% RSLogix 500 project I2P JOB 12 B ALEXANDER_LOYND_BAK034.RSS, saved by version 10.00.00.00 %
PROJECT "ML06A"    % processor: Bul.1763 MicroLogix 1100 Series B %

PROGRAM FILES
  LAD 2   13 rungs

DATA FILES
  O0 OUTPUT  4 elements
  I1 INPUT  6 elements
  S2 STATUS  66 elements
  B3 BINARY  1 elements
  T4 TIMER  1 elements
  C5 COUNTER  1 elements
  R6 CONTROL  1 elements
  N7 INTEGER  1 elements
  F8 FLOAT  1 elements

LADDER 2
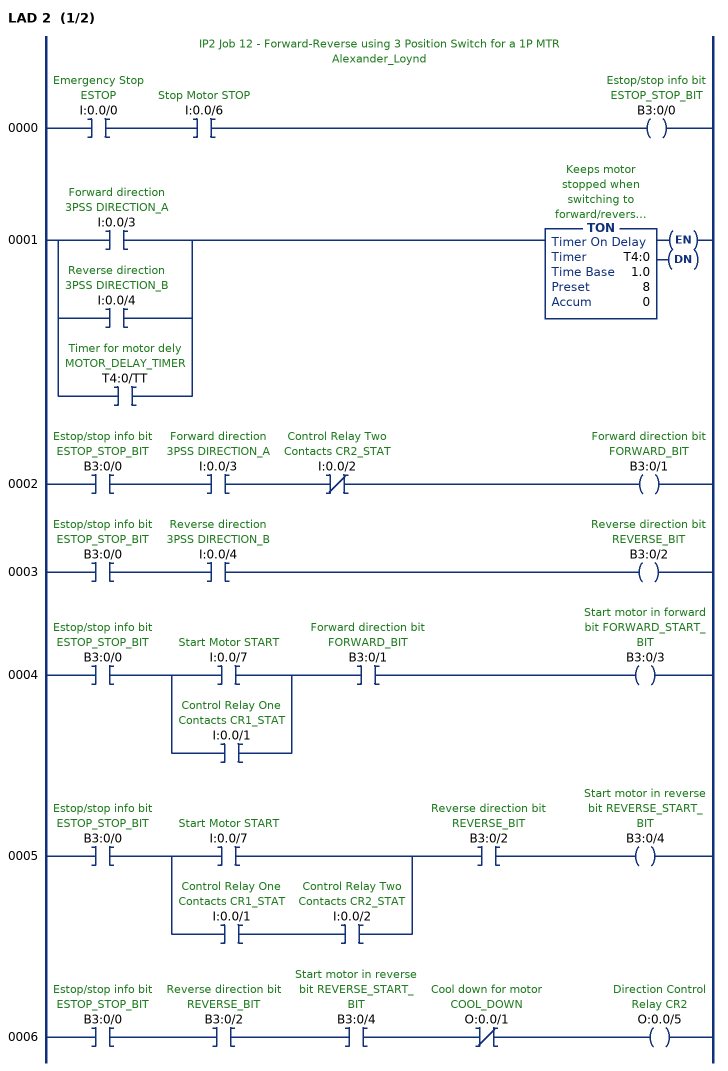
% Rung: 0 %
% IP2 Job 12 - Forward-Reverse using 3 Position Switch for a 1P MTR
% Alexander_Loynd %
SOR XIC I:0.0/0 XIC I:0.0/6 OTE B3:0/0 EOR
%   I:0.0/0  ESTOP  "Emergency Stop" %
%   I:0.0/6  STOP  "Stop Motor" %
%   B3:0/0  ESTOP_STOP_BIT  "Estop/stop info bit" %
% Rung: 1 %
SOR BST XIC I:0.0/3 NXB BST XIC I:0.0/4 NXB XIC T4:0/TT BND BND TON T4:0 1.0 8 0 EOR
%   I:0.0/3  DIRECTION_A  "Forward direction 3PSS" %
%   I:0.0/4  DIRECTION_B  "Reverse direction 3PSS" %
%   T4:0/TT  MOTOR_DELAY_TIMER  "Timer for motor dely" %
%   T4:0  TIME_ON_DELAY  "Keeps motor stopped when switching to forward/reverse" %
% Rung: 2 %
SOR XIC B3:0/0 XIC I:0.0/3 XIO I:0.0/2 OTE B3:0/1 EOR
%   B3:0/0  ESTOP_STOP_BIT  "Estop/stop info bit" %
%   I:0.0/3  DIRECTION_A  "Forward direction 3PSS" %
%   I:0.0/2  CR2_STAT  "Control Relay Two Contacts" %
%   B3:0/1  FORWARD_BIT  "Forward direction bit" %
% Rung: 3 %
SOR XIC B3:0/0 XIC I:0.0/4 OTE B3:0/2 EOR
%   B3:0/0  ESTOP_STOP_BIT  "Estop/stop info bit" %
%   I:0.0/4  DIRECTION_B  "Reverse direction 3PSS" %
%   B3:0/2  REVERSE_BIT  "Reverse direction bit" %
% Rung: 4 %
SOR XIC B3:0/0 BST XIC I:0.0/7 NXB XIC I:0.0/1 BND XIC B3:0/1 OTE B3:0/3 EOR
%   B3:0/0  ESTOP_STOP_BIT  "Estop/stop info bit" %
%   I:0.0/7  START  "Start Motor" %
%   I:0.0/1  CR1_STAT  "Control Relay One Contacts" %
%   B3:0/1  FORWARD_BIT  "Forward direction bit" %
%   B3:0/3  FORWARD_START_BIT  "Start motor in forward bit" %
% Rung: 5 %
SOR XIC B3:0/0 BST XIC I:0.0/7 NXB XIC I:0.0/1 XIC I:0.0/2 BND XIC B3:0/2 OTE B3:0/4 EOR
%   B3:0/0  ESTOP_STOP_BIT  "Estop/stop info bit" %
%   I:0.0/7  START  "Start Motor" %
%   I:0.0/1  CR1_STAT  "Control Relay One Contacts" %
%   I:0.0/2  CR2_STAT  "Control Relay Two Contacts" %
%   B3:0/2  REVERSE_BIT  "Reverse direction bit" %
%   B3:0/4  REVERSE_START_BIT  "Start motor in reverse bit" %
% Rung: 6 %
SOR XIC B3:0/0 XIC B3:0/2 XIC B3:0/4 XIO O:0.0/1 OTE O:0.0/5 EOR
%   B3:0/0  ESTOP_STOP_BIT  "Estop/stop info bit" %
%   B3:0/2  REVERSE_BIT  "Reverse direction bit" %
%   B3:0/4  REVERSE_START_BIT  "Start motor in reverse bit" %
%   O:0.0/1  COOL_DOWN  "Cool down for motor" %
%   O:0.0/5  CR2  "Direction Control Relay" %

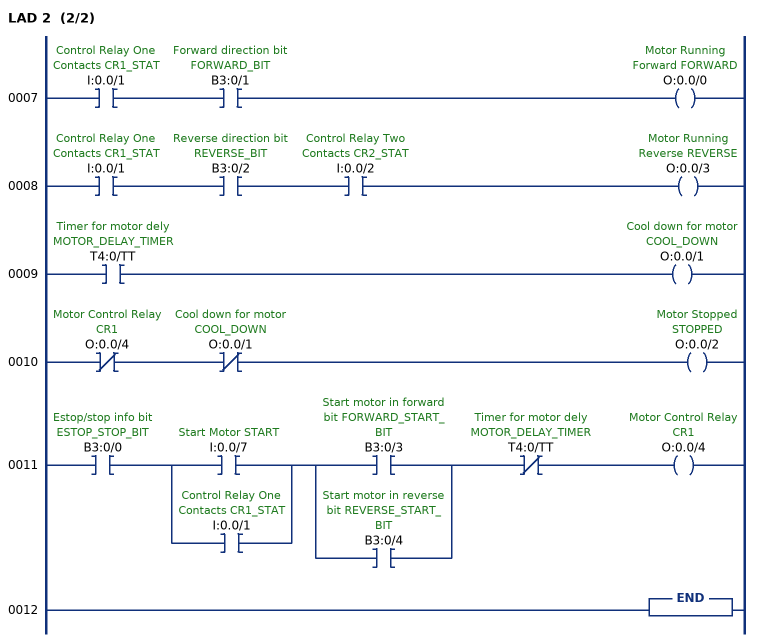
% Rung: 7 %
SOR XIC I:0.0/1 XIC B3:0/1 OTE O:0.0/0 EOR
%   I:0.0/1  CR1_STAT  "Control Relay One Contacts" %
%   B3:0/1  FORWARD_BIT  "Forward direction bit" %
%   O:0.0/0  FORWARD  "Motor Running Forward" %
% Rung: 8 %
SOR XIC I:0.0/1 XIC B3:0/2 XIC I:0.0/2 OTE O:0.0/3 EOR
%   I:0.0/1  CR1_STAT  "Control Relay One Contacts" %
%   B3:0/2  REVERSE_BIT  "Reverse direction bit" %
%   I:0.0/2  CR2_STAT  "Control Relay Two Contacts" %
%   O:0.0/3  REVERSE  "Motor Running Reverse" %
% Rung: 9 %
SOR XIC T4:0/TT OTE O:0.0/1 EOR
%   T4:0/TT  MOTOR_DELAY_TIMER  "Timer for motor dely" %
%   O:0.0/1  COOL_DOWN  "Cool down for motor" %
% Rung: 10 %
SOR XIO O:0.0/4 XIO O:0.0/1 OTE O:0.0/2 EOR
%   O:0.0/4  CR1  "Motor Control Relay" %
%   O:0.0/1  COOL_DOWN  "Cool down for motor" %
%   O:0.0/2  STOPPED  "Motor Stopped" %
% Rung: 11 %
SOR XIC B3:0/0 BST XIC I:0.0/7 NXB XIC I:0.0/1 BND BST XIC B3:0/3 NXB XIC B3:0/4 BND XIO T4:0/TT OTE O:0.0/4 EOR
%   B3:0/0  ESTOP_STOP_BIT  "Estop/stop info bit" %
%   I:0.0/7  START  "Start Motor" %
%   I:0.0/1  CR1_STAT  "Control Relay One Contacts" %
%   B3:0/3  FORWARD_START_BIT  "Start motor in forward bit" %
%   B3:0/4  REVERSE_START_BIT  "Start motor in reverse bit" %
%   T4:0/TT  MOTOR_DELAY_TIMER  "Timer for motor dely" %
%   O:0.0/4  CR1  "Motor Control Relay" %
% Rung: 12 %
SOR END EOR

OTHER DOCUMENTED ADDRESSES
  I:0.0/5  2PSS  "Two Position Selector Switch"
  I:0.0/8  PB3  "Push Button, NO"
  PB1  "Start Motor"

DATA TABLE (non-zero values as saved)
DATA T4
% .PRE .ACC %
% T4:0 % 8 0
